(* IEC 61131-3 sources: F100R_S278_Temperville/MyController.device.xml.v3^/Plc Logic.plclogic.xml.v3^/Application.application.xml.v3^/07_Energia, 9 files *)

(* ---- C_ComposicaoFatura.prg.st ---- *)
PROGRAM C_ComposicaoFatura
VAR
	TonHabilita: TON;
	xTonHabilitaIn: BOOL;
	xTonHabilitaQ: BOOL;
	xTonHabilitaPt: TIME;
	PulsoLeitura: PulsoPositivo;
	PulsoLeituraIn: BOOL;
	PulsoLeituraQ: BOOL;
	xIntervaloPonta: BOOL;
	xIntervaloFPonta: BOOL;
	xIntervaloFPonta01: BOOL;
	xIntervaloFPonta02: BOOL;
	xFimMes: BOOL;
	xFechaConta: BOOL;
	rDemandaInstantaneaReal_kW: REAL;
END_VAR

(*LÓGICA DE COMPOSIÇÃO DA FATURA DE ENERGIA E ZERAMENTO DO MEDIDOR*)

// Dia da Leitura -> Fecha Fatura

IF uDiadaLeitura=uDiaRealTime THEN
	PulsoLeituraIn:=TRUE;
ELSE
	PulsoLeituraIn:=FALSE;
END_IF

PulsoLeitura(Entrada:=PulsoLeituraIn , SaidaPulsoPo=>PulsoLeituraQ );

IF PulsoLeituraQ THEN
	xFimMes:=TRUE;
END_IF

IF xFimMes THEN
	xFechaFatura:=1;
	xFimMes:=FALSE;
END_IF

(*-------------------------------------------------------------------------*)
xTonHabilitaIn:=TRUE;
TonHabilita(IN:=xTonHabilitaIn , PT:=T#300MS(*xTonHabilitaPt*) , Q=> xTonHabilitaQ, ET=> );

(*========= INTERVALOS DE PONTA E FORA PONTA =========*)

IF uHoraRealTime>=uHoraPonta  AND uHoraRealTime<=uHoraFPonta THEN
	xIntervaloPonta:=TRUE;
	xIntervaloFPonta:=FALSE;
ELSE
	xIntervaloFPonta:=TRUE;
	xIntervaloPonta:=FALSE;
END_IF

CASE PassoIntervalo OF
	//Seleção do Intervalo
		0: 	IF xIntervaloFPonta AND xTonHabilitaQ THEN
				PassoIntervalo:=5;
			END_IF
			IF xIntervaloPonta AND xTonHabilitaQ THEN
				PassoIntervalo:=50;
			END_IF
	// Consumos Fora Ponta
		5:	rConsumoInicialFPonta_kW:=rConsumoEnergiaReal_kWh;(*Ativo*)
			rConsumoInicialFPonta_kVAR:=rConsumoEnergiaReativa_kVARh;(*Reativo*)
			PassoIntervalo:=10;

		10:	rConsumoInstantaneoFPonta_kW:=rConsumoEnergiaReal_kWh-rConsumoInicialFPonta_kW;(*Ativo*)
			rConsumoInstantAcumFPonta_kW:=rConsumoAcumuladoFPonta_kW+rConsumoInstantaneoFPonta_kW;(*Ativo*)
			rConsumoInstantaneoFPonta_kVAR:=rConsumoEnergiaReativa_kVARh-rConsumoInicialFPonta_kVAR;(*Reativo*)
			rConsumoInstantAcumFPonta_kVAR:=rConsumoAcumuladoFPonta_kVAR+rConsumoInstantaneoFPonta_kVAR;(*Reativo*)

			rDemandaInstantaneaReal_kW:=rDemandaTotalReal_kW;
			IF rDemandaInstantaneaReal_kW>rDemandaMaximaPeriodo_kW THEN
				rDemandaMaximaPeriodo_kW:=rDemandaInstantaneaReal_kW;
			END_IF

			IF rDemandaTotalReal_kW>rDemandaMaximaIntervalo THEN
				rDemandaMaximaIntervalo:=rDemandaTotalReal_kW;
			END_IF

			IF NOT xIntervaloFPonta AND xTonHabilitaQ THEN
				PassoIntervalo:=15;
			END_IF
			IF (xFechaFatura=1) AND xTonHabilitaQ THEN
				PassoIntervalo:=16;
			END_IF

		15:	rConsumoAcumuladoFPonta_kW:=rConsumoInstantAcumFPonta_kW;(*Ativo*)
			rConsumoAcumuladoFPonta_kVAR:=rConsumoInstantAcumFPonta_kVAR;(*Reativo*)
			rConsumoFPonta_kW:=rConsumoInstantaneoFPonta_kW;(*Ativo*)
			rConsumoFPonta_kVAR:=rConsumoInstantaneoFPonta_kVAR;(*Reativo*)
			rDemandaMaxUltimoPeriodo:=rDemandaMaximaPeriodo_kW;
			PassoIntervalo:=16;

		16:	PassoIntervalo:=20;

		18: rConsumoAcumuladoFPonta_kW:=rConsumoInstantAcumFPonta_kW;(*Ativo*)
			rConsumoAcumuladoFPonta_kVAR:=rConsumoInstantAcumFPonta_kVAR;(*Reativo*)
			rConsumoFPonta_kW:=rConsumoInstantaneoFPonta_kW;(*Ativo*)
			rConsumoFPonta_kVAR:=rConsumoInstantaneoFPonta_kVAR;(*Reativo*)
			//rDemandaMaxUltimoIntervalo:=rDemandaMaximaReal_kW;
			rDemandaMaxUltimoIntervalo:=rDemandaMaximaIntervalo;
			PassoIntervalo:=20;

		20:	rConsumoInstantaneoFPonta_kW:=0;(*Ativo*)
			rConsumoInstantaneoFPonta_kVAR:=0;(*Reativo*)
			rDemandaMaximaPeriodo_kW:=0;
			IF (xFechaFatura=1) THEN
				xFechaConta:=TRUE;
			END_IF
			PassoIntervalo:=0;
	// Consumos Ponta
		50:	rConsumoInicialPonta_kW:=rConsumoEnergiaReal_kWh;(*Ativo*)
			rConsumoInicialPonta_kVAR:=rConsumoEnergiaReativa_kVARh;(*Reativo*)
			PassoIntervalo:=55;

		55:	rConsumoInstantaneoPonta_kW:=rConsumoEnergiaReal_kWh-rConsumoInicialPonta_kW;(*Ativo*)
			rConsumoInstantAcumPonta_kW:=rConsumoAcumuladoPonta_kW+rConsumoInstantaneoPonta_kW;(*Ativo*)
			rConsumoInstantaneoPonta_kVAR:=rConsumoEnergiaReativa_kVARh-rConsumoInicialPonta_kVAR;(*Reativo*)
			rConsumoInstantAcumPonta_kVAR:=rConsumoAcumuladoPonta_kVAR+rConsumoInstantaneoPonta_kVAR;(*Reativo*)

			rDemandaInstantaneaReal_kW:=rDemandaTotalReal_kW;
			IF rDemandaInstantaneaReal_kW>rDemandaMaximaPeriodo_kW THEN
				rDemandaMaximaPeriodo_kW:=rDemandaInstantaneaReal_kW;
			END_IF

			IF rDemandaTotalReal_kW>rDemandaMaximaIntervalo THEN
				rDemandaMaximaIntervalo:=rDemandaTotalReal_kW;
			END_IF

			IF NOT xIntervaloPonta AND xTonHabilitaQ THEN
				PassoIntervalo:=60;
			END_IF
			IF (xFechaFatura=1) AND xTonHabilitaQ THEN
				PassoIntervalo:=61;
			END_IF

		60:	rConsumoPonta_kW:=rConsumoInstantaneoPonta_kW;(*Ativo*)
			rConsumoAcumuladoPonta_kW:=rConsumoInstantAcumPonta_kW;(*Ativo*)
	      	rConsumoPonta_kVAR:=rConsumoInstantaneoPonta_kVAR;(*Reativo*)
			rConsumoAcumuladoPonta_kVAR:=rConsumoInstantAcumPonta_kVAR;(*Reativo*)
			rDemandaMaxUltimoPeriodo:=rDemandaMaximaPeriodo_kW;
			PassoIntervalo:=61;

		61:	PassoIntervalo:=65;

		63:	rConsumoPonta_kW:=rConsumoInstantaneoPonta_kW;(*Ativo*)
			rConsumoAcumuladoPonta_kW:=rConsumoInstantAcumPonta_kW;(*Ativo*)
	      	rConsumoPonta_kVAR:=rConsumoInstantaneoPonta_kVAR;(*Reativo*)
			rConsumoAcumuladoPonta_kVAR:=rConsumoInstantAcumPonta_kVAR;(*Reativo*)
			//rDemandaMaxUltimoIntervalo:=rDemandaMaximaReal_kW;
			rDemandaMaxUltimoIntervalo:=rDemandaMaximaIntervalo;
			PassoIntervalo:=65;

		65:	rConsumoInstantaneoPonta_kW:=0;(*Ativo*)
			rConsumoInstantaneoPonta_kVAR:=0;(*Reativo*)
			rDemandaMaximaPeriodo_kW:=0;
			IF (xFechaFatura=1) THEN
				xFechaConta:=TRUE;
			END_IF
			PassoIntervalo:=0;
END_CASE

// Fechamento da Tarifa Mensal
IF xFechaConta AND xTonHabilitaQ THEN
	 rEnergiaAtivaPonta_kWh			:=rConsumoAcumuladoPonta_kW;
	 rEnergiaAtivaFPonta_kWh		:=rConsumoAcumuladoFPonta_kW;
	 rEnergiaReativaPonta_kVar		:=rConsumoAcumuladoPonta_kVAR;
	 rEnergiaReativaFPonta_kVar		:=rConsumoAcumuladoFPonta_kVAR;
	 rDemandaEnergia_kW				:=rDemandaMaxUltimoIntervalo;
	 xFechaConta:=FALSE;
END_IF

IF xFaturaFechada=1 THEN // Vem do Supervisório
	bZeraAcumulado		:=TRUE;
	xCmdResetGeralPm	:=TRUE;
	xFaturaFechada		:=0;
END_IF

(*--------------------------------------------------------------------------------------------------------
(*--------------- Consumo Intervalo Diario -------*)
(*========= INTERVALOS FORA PONTA 01 e 02 =========*)

IF uMinutoRealTime>=0 AND uMinutoRealTime<=uMinutoPonta THEN
	xIntervaloFPonta01:=TRUE;
	xIntervaloFPonta02:=FALSE;
ELSIF uMinutoRealTime>=uMinutoFPonta AND  uMinutoRealTime<59 THEN
	xIntervaloFPonta02:=TRUE;
	xIntervaloFPonta01:=FALSE;
ELSIF uMinutoRealTime>=uMinutoPonta AND uMinutoRealTime<=uMinutoFPonta THEN
	xIntervaloFPonta01:=FALSE;
	xIntervaloFPonta02:=FALSE;
END_IF

CASE PassoIntervaloDia OF

		0: 	IF xIntervaloFPonta01 AND xTonHabilitaQ THEN
				PassoIntervaloDia:=5;
			END_IF
			IF xIntervaloFPonta02 AND xTonHabilitaQ THEN
				PassoIntervaloDia:=50;
			END_IF

		5:	rConsumoInicialFPonta01:=rConsumoEnergiaReal_kWh;
			PassoIntervaloDia:=10;

		10:	rConsumoInstantaneoFPonta01:=rConsumoEnergiaReal_kWh-rConsumoInicialFPonta01;
			rConsumoInstantDiarioFPonta:=rConsumoInstantaneoFPonta01;
			IF NOT xIntervaloFPonta01 AND xTonHabilitaQ THEN
				PassoIntervaloDia:=15;
			END_IF

		15:	rConsumoFPonta01:=rConsumoInstantaneoFPonta01;
			PassoIntervaloDia:=20;

		20:	rConsumoInstantaneoFPonta01:=0;
			PassoIntervaloDia:=0;

		50:	rConsumoInicialFPonta02:=rConsumoEnergiaReal_kWh;
			PassoIntervaloDia:=55;

		55:	rConsumoInstantaneoFPonta02:=rConsumoEnergiaReal_kWh-rConsumoInicialFPonta02;
			rConsumoInstantDiarioFPonta:=rConsumoFPonta01+rConsumoInstantaneoFPonta02;
			IF NOT xIntervaloFPonta02 AND xTonHabilitaQ THEN
				PassoIntervaloDia:=60;
			END_IF

		60:	rConsumoFPonta02:=rConsumoInstantaneoFPonta02;
			PassoIntervaloDia:=65;

		65:	rConsumoInstantaneoFPonta02:=0;
			rConsumoInstantDiarioFPonta:=0;
			PassoIntervaloDia:=70;

		70:	rConsumoDiarioFPonta:=rConsumoFPonta01+rConsumoFPonta02;
			rConsumoInicialFPonta01:=0;
			rConsumoInstantaneoFPonta01:=0;
			rConsumoFPonta01:=0;
			rConsumoInicialFPonta02:=0;
			rConsumoInstantaneoFPonta02:=0;
			rConsumoFPonta02:=0;
			PassoIntervaloDia:=0;

END_CASE
---------------------------------------------------------------------------------------------------------------*)
// ENERGIA CONSUMO DIÁRIO

rConsumoDiario:= rConsumoEnergiaReal_kWh-rConsumoDiarioInicial_kW;

IF	(uHoraRealTime=23 AND uMinutoRealTime=59 AND uSegundoRealTime=0) THEN
	rConsumoDiarioRel:=rConsumoDiario;
	xGrvRelatorioEnerg:=TRUE;

END_IF

IF	(uHoraRealTime=0 AND uMinutoRealTime=0 AND uSegundoRealTime=0)  THEN
	rConsumoDiarioInicial_kW:=rConsumoEnergiaReal_kWh;

END_IF

(* ---- D_ZeramentoMedidor.prg.st ---- *)
PROGRAM D_ZeramentoMedidor
VAR
	///Passo da Execução Reset Medidor de Energia
	PassoResetPm: INT;
	uResetValoresPM: UINT;
	xTriggerResetPM: BOOL;
	TonReset: TON;
	xTonResetIn: BOOL;
	xTonResetQ: BOOL;
	xTonResePt: TIME := TIME#2s0ms;
END_VAR

//Zeramento do Valores do Medidor
CASE PassoResetPm OF

		0:	IF xCmdResetGeralPm THEN
				uResetValoresPM:=14255;
				PassoResetPm:=1;
			END_IF

		1: IF uResetValoresPM=14255 THEN
				PassoResetPm:=3;
			END_IF

		3:	xTonResetIn:=TRUE;
			IF	xTonResetQ THEN
					PassoResetPm:=5;
			END_IF

		5:	xTonResetIn:=FALSE;
			xTriggerResetPM:=TRUE;
			PassoResetPm:=7;

		7:	xTonResetIn:=TRUE;
			IF	xTonResetQ THEN
					PassoResetPm:=10;
			END_IF

		10: xTonResetIn:=FALSE;
			xTriggerResetPM:=FALSE;
			uResetValoresPM:=30078;
			PassoResetPm:=11;

		11: IF uResetValoresPM=30078 THEN
				PassoResetPm:=13;
			END_IF

		13:	xTonResetIn:=TRUE;
			IF	xTonResetQ THEN
					PassoResetPm:=15;
			END_IF

		15:	xTonResetIn:=FALSE;
			xTriggerResetPM:=TRUE;
			PassoResetPm:=17;

		17:	xTonResetIn:=TRUE;
			IF	xTonResetQ AND rConsumoEnergiaReal_kWh=0 THEN
					PassoResetPm:=20;
			END_IF

		20:	xTonResetIn:=FALSE;
			xTriggerResetPM:=FALSE;
			uResetValoresPM:=21212;
			PassoResetPm:=21;

		21: IF uResetValoresPM=21212 THEN
				PassoResetPm:=23;
			END_IF

		23:	xTonResetIn:=TRUE;
			IF	xTonResetQ THEN
					PassoResetPm:=25;
			END_IF

		25:	xTonResetIn:=FALSE;
			xTriggerResetPM:=TRUE;
			PassoResetPm:=27;

		27:	xTonResetIn:=TRUE;
			IF	xTonResetQ THEN
					PassoResetPm:=30;
			END_IF

		30:	xTonResetIn:=FALSE;
			xTriggerResetPM:=FALSE;
			uResetValoresPM:=10001;
			PassoResetPm:=31;

		31: IF uResetValoresPM=10001 THEN
				PassoResetPm:=33;
			END_IF

		33:	xTonResetIn:=TRUE;
			IF	xTonResetQ THEN
					PassoResetPm:=35;
			END_IF

		35:	xTonResetIn:=FALSE;
			xTriggerResetPM:=TRUE;
			PassoResetPm:=37;

		37:	xTonResetIn:=TRUE;
			IF	xTonResetQ THEN
					PassoResetPm:=40;
			END_IF

		40:	xTonResetIn:=FALSE;
			xTriggerResetPM:=FALSE;
			uResetValoresPM:=0;
			bZeraAcumulado:=TRUE;
			xCmdResetGeralPm:=FALSE;
			PassoResetPm:=0;

END_CASE
TonReset(IN:= xTonResetIn, PT:=T#2S(*xTonResePt*) , Q=> xTonResetQ, ET=> );

// Zeramento das Memorias Acumuladas
IF bZeraAcumulado THEN
	PassoIntervalo				:=0;

	rConsumoInicialFPonta_kW	:=0;
	rConsumoInstantaneoFPonta_kW:=0;
	rConsumoFPonta_kW			:=0;
	rConsumoInstantAcumFPonta_kW:=0;
	rConsumoAcumuladoFPonta_kW	:=0;

	rConsumoInicialPonta_kW		:=0;
	rConsumoInstantaneoPonta_kW	:=0;
	rConsumoPonta_kW			:=0;
	rConsumoInstantAcumPonta_kW	:=0;
	rConsumoAcumuladoPonta_kW	:=0;

	rConsumoInicialFPonta_kVAR	:=0;
	rConsumoInstantaneoFPonta_kVAR:=0;
	rConsumoFPonta_kVAR			:=0;
	rConsumoInstantAcumFPonta_kVAR:=0;
	rConsumoAcumuladoFPonta_kVAR:=0;

	rConsumoInicialPonta_kVAR	:=0;
	rConsumoInstantaneoPonta_kVAR:=0;
	rConsumoPonta_kVAR			:=0;
	rConsumoInstantAcumPonta_kVAR:=0;
	rConsumoAcumuladoPonta_kVAR	:=0;

//	rConsumoInicialFPonta01		:=0;
//	rConsumoInstantaneoFPonta01	:=0;
//	rConsumoFPonta01			:=0;

//	rConsumoInicialFPonta02		:=0;
//	rConsumoInstantaneoFPonta02	:=0;
//	rConsumoFPonta02			:=0;

	rConsumoDiarioFPonta		:=0;
	//xFaturaFechada				:=0;
	bZeraAcumulado				:=FALSE;
END_IF

(* ---- E_Nobreak.prg.st ---- *)
PROGRAM E_Nobreak
VAR
	TonNobreak: TON;
	TonNobreakIn: BOOL;
	TonNobreakQ: BOOL;
	TpSonAlmNbk: TP;
END_VAR

xStatusNobreak:=xSaidaNobreakOk;

TonNobreakIn:= NOT xSaidaNobreakOk;
TonNobreak(IN:=TonNobreakIn , PT:=T#500MS , Q=>TonNobreakQ , ET=> );
IF TonNobreakQ THEN
	xAlmNobreak:=TRUE;
END_IF

TpSonAlmNbk(IN:=xAlmNobreak , PT:=T#500MS , Q=> , ET=> );

IF TpSonAlmNbk.Q THEN
	xAlmNobreakSom:=TRUE;
END_IF

IF	bResetAlmGeral THEN
	xAlmNobreak:=FALSE;
	xAlmNobreakSom:=FALSE;
END_IF

xNobreakDesabilitado:= NOT xNobreakHabilitado;

(* ---- Energia.prg.st ---- *)
PROGRAM Energia
VAR
	Double01: WORD_AS_DWORD;
	Double02: WORD_AS_DWORD;
	Double03: WORD_AS_DWORD;
	////////////////////////////////////////////////////////////////
	dConsumoEnergiaReal_kWh: DWORD;
	dConsumoEnergiaAparente_kVAh: DWORD;
	dConsumoEnergiaReativa_kVARh: DWORD;
	u0ConsumoEnergiaReal_kWh: WORD;
	u1ConsumoEnergiaReal_kWh: WORD;
	u0ConsumoEnergiaAparente_kVAh: WORD;
	u1ConsumoEnergiaAparente_kVAh: WORD;
	u0ConsumoEnergiaReativa_kVARh: WORD;
	u1ConsumoEnergiaReativa_kVARh: WORD;
	uPotenciaTotalReal_kW: UINT;
	uPotenciaTotalAparente_kVA: UINT;
	uPotenciaTotalReativa_kVAR: UINT;
	uFatorDePotenciaTotal: UINT;
	uTensaoFFMedia_V: UINT;
	uTensaoFNMedia_V: UINT;
	uCorrenteMedia_V: UINT;
	uFrequencia_Hz: UINT;
	uDemandaTotalReal_kW: UINT;
	uDemandaTotalAparente_kVA: UINT;
	uDemandaTotalReativa_kVAR: UINT;
	uDemandaMaximaReal_kW: UINT;
	uDemandaMaximaAparente_kVA: UINT;
	uDemandaMaximaReativa_kVAR: UINT;
	uCorrenteInstantFaseA_Amp: UINT;
	uCorrenteInstantFaseB_Amp: UINT;
	uCorrenteInstantFaseC_Amp: UINT;
	uCorrenteInstantNeutro_Amp: UINT;
	uCorrenteDemandaFaseA_Amp: UINT;
	uCorrenteDemandaFaseB_Amp: UINT;
	uCorrenteDemandaFaseC_Amp: UINT;
	uCorrenteMaximaDemandaFaseA_Amp: UINT;
	uCorrenteMaximaDemandaFaseB_Amp: UINT;
	uCorrenteMaximaDemandaFaseC_Amp: UINT;
	uTensaoFaseAB_V: UINT;
	uTensaoFaseBC_V: UINT;
	uTensaoFaseAC_V: UINT;
	uTensaoFaseAN_V: UINT;
	uTensaoFaseBN_V: UINT;
	uTensaoFaseCN_V: UINT;
	uPotenciaRealFaseA_kW: UINT;
	uPotenciaRealFaseB_kW: UINT;
	uPotenciaRealFaseC_kW: UINT;
	uPotenciaAparenteFaseA_kVA: UINT;
	uPotenciaAparenteFaseB_kVA: UINT;
	uPotenciaAparenteFaseC_kVA: UINT;
	uPotenciaReativaFaseA_kVAR: UINT;
	uPotenciaReativaFaseB_kVAR: UINT;
	uPotenciaReativaFaseC_kVAR: UINT;
	uCorrenteTHDFaseA: UINT;
	uCorrenteTHDFaseB: UINT;
	uCorrenteTHDFaseC: UINT;
	uCorrenteTHDNeutro: UINT;
	uTensaoTHDFaseAN: UINT;
	uTensaoTHDFaseBN: UINT;
	uTensaoTHDFaseCN: UINT;
	uTensaoTHDFaseAB: UINT;
	uTensaoTHDFaseBC: UINT;
	uTensaoTHDFaseAC: UINT;
	/// Valores minimos
	uPotenciaTotalRealMinima_kW: UINT;
	uPotenciaTotalAparenteMinima_kVA: UINT;
	uPotenciaTotalReativaMinima_kVAR: UINT;
	uFatorDePotenciaTotalMinima: UINT;
	uFrequenciaMinima_Hz: UINT;
	uCorrenteMinimaFaseA_Amp: UINT;
	uCorrenteMinimaFaseB_Amp: UINT;
	uCorrenteMinimaFaseC_Amp: UINT;
	uCorrenteMinimaNeutro_Amp: UINT;
	uTensaoMinimaFaseAN_V: UINT;
	uTensaoMinimaFaseBN_V: UINT;
	uTensaoMinimaFaseCN_V: UINT;
	uTensaoMinimaFaseAB_V: UINT;
	uTensaoMinimaFaseBC_V: UINT;
	uTensaoMinimaFaseAC_V: UINT;
	uCorrenteTHDMinimoFaseA: UINT;
	uCorrenteTHDMinimoFaseB: UINT;
	uCorrenteTHDMinimoFaseC: UINT;
	uCorrenteTHDMinimoNeutro: UINT;
	uTensaoTHDMinimoFaseAN: UINT;
	uTensaoTHDMinimoFaseBN: UINT;
	uTensaoTHDMinimoFaseCN: UINT;
	uTensaoTHDMinimoFaseAB: UINT;
	uTensaoTHDMinimoFaseBC: UINT;
	uTensaoTHDMinimoFaseAC: UINT;
	/// Valores Maximos
	uPotenciaTotalRealMaximo_kW: UINT;
	uPotenciaTotalAparenteMaximo_kVA: UINT;
	uPotenciaTotalReativaMaximo_kVAR: UINT;
	uFatorDePotenciaTotalMaximo: UINT;
	uFrequenciaMaxima_Hz: UINT;
	uCorrenteMaximoFaseA_Amp: UINT;
	uCorrenteMaximoFaseB_Amp: UINT;
	uCorrenteMaximoFaseC_Amp: UINT;
	uCorrenteMaximoNeutro_Amp: UINT;
	uTensaoMaximoFaseAN_V: UINT;
	uTensaoMaximoFaseBN_V: UINT;
	uTensaoMaximoFaseCN_V: UINT;
	uTensaoMaximoFaseAB_V: UINT;
	uTensaoMaximoFaseBC_V: UINT;
	uTensaoMaximoFaseAC_V: UINT;
	uCorrenteTHDMaximoFaseA: UINT;
	uCorrenteTHDMaximoFaseB: UINT;
	uCorrenteTHDMaximoFaseC: UINT;
	uCorrenteTHDMaximoNeutro: UINT;
	uTensaoTHDMaximoFaseAN: UINT;
	uTensaoTHDMaximoFaseBN: UINT;
	uTensaoTHDMaximoFaseCN: UINT;
	uTensaoTHDMaximoFaseAB: UINT;
	uTensaoTHDMaximoFaseBC: UINT;
	uTensaoTHDMaximoFaseAC: UINT;
END_VAR

Double01(i_wLow:= u1ConsumoEnergiaReal_kWh, i_wHigh:= u0ConsumoEnergiaReal_kWh, q_dwOput=> dConsumoEnergiaReal_kWh);
Double02(i_wLow:= u1ConsumoEnergiaAparente_kVAh, i_wHigh:= u0ConsumoEnergiaAparente_kVAh, q_dwOput=> dConsumoEnergiaAparente_kVAh);
Double03(i_wLow:= u1ConsumoEnergiaReativa_kVARh, i_wHigh:= u0ConsumoEnergiaReativa_kVARh, q_dwOput=> dConsumoEnergiaReativa_kVARh);

rConsumoEnergiaReal_kWh			:=fEnergiaAtivaAcumulada/1000;//(DINT_TO_REAL(DWORD_TO_DINT(dConsumoEnergiaReal_kWh)))/10;
rConsumoEnergiaAparente_kVAh	:=fEnergiaAparenteAcumulada/1000;//(DINT_TO_REAL(DWORD_TO_DINT(dConsumoEnergiaAparente_kVAh)))/10;
rConsumoEnergiaReativa_kVARh	:=fEnergiaReativaAcumulada/1000;//(DINT_TO_REAL(DWORD_TO_DINT(dConsumoEnergiaReativa_kVARh)))/10;
rPotenciaTotalReal_kW			:=fPotenciaAtivaTotal;//(INT_TO_REAL(UINT_TO_INT(uPotenciaTotalReal_kW)));
rPotenciaTotalAparente_kVA		:=(INT_TO_REAL(UINT_TO_INT(uPotenciaTotalAparente_kVA)));
rPotenciaTotalReativa_kVAR 		:=(INT_TO_REAL(UINT_TO_INT(uPotenciaTotalReativa_kVAR)))/10;
rFatorDePotenciaTotal 			:=fFatorPotenciaTotal;//(INT_TO_REAL(UINT_TO_INT(uFatorDePotenciaTotal)))/10000;
rTensaoFFMedia_V				:=fTensaoAvgLL;//(INT_TO_REAL(UINT_TO_INT(uTensaoFFMedia_V)))/10;
rTensaoFNMedia_V				:=fTensaoAvgLN;//(INT_TO_REAL(UINT_TO_INT(uTensaoFNMedia_V)))/10;
rCorrenteMedia_V				:=fCorrenteAvg;//(INT_TO_REAL(UINT_TO_INT(uCorrenteMedia_V)));
rFrequencia_Hz					:=fFrequencia;//(INT_TO_REAL(UINT_TO_INT(uFrequencia_Hz)))/100;
rDemandaTotalReal_kW			:=fUltimaDemanda;//(INT_TO_REAL(UINT_TO_INT(uDemandaTotalReal_kW)));
rDemandaTotalAparente_kVA		:=(INT_TO_REAL(UINT_TO_INT(uDemandaTotalAparente_kVA)));
rDemandaTotalReativa_kVAR		:=(INT_TO_REAL(UINT_TO_INT(uDemandaTotalReativa_kVAR)))/10;
rDemandaMaximaReal_kW			:=fPicoDemanda;//(INT_TO_REAL(UINT_TO_INT(uDemandaMaximaReal_kW)));
rDemandaMaximaAparente_kVA		:=(INT_TO_REAL(UINT_TO_INT(uDemandaMaximaAparente_kVA)))/10;
rDemandaMaximaReativa_kVAR		:=(INT_TO_REAL(UINT_TO_INT(uDemandaMaximaReativa_kVAR)))/10;
rCorrenteInstantFaseA_Amp		:=fCorrenteFaseA;//(INT_TO_REAL(UINT_TO_INT(uCorrenteInstantFaseA_Amp)))/1;
rCorrenteInstantFaseB_Amp 		:=fCorrenteFaseB;//(INT_TO_REAL(UINT_TO_INT(uCorrenteInstantFaseB_Amp)))/1;
rCorrenteInstantFaseC_Amp 		:=fCorrenteFaseC;//(INT_TO_REAL(UINT_TO_INT(uCorrenteInstantFaseC_Amp)))/1;
rCorrenteInstantNeutro_Amp 		:=fCorrenteNeutro;//(INT_TO_REAL(UINT_TO_INT(uCorrenteInstantNeutro_Amp)))/1;
rCorrenteDemandaFaseA_Amp		:=(INT_TO_REAL(UINT_TO_INT(uCorrenteDemandaFaseA_Amp)))/10;
rCorrenteDemandaFaseB_Amp		:=(INT_TO_REAL(UINT_TO_INT(uCorrenteDemandaFaseB_Amp)))/10;
rCorrenteDemandaFaseC_Amp		:=(INT_TO_REAL(UINT_TO_INT(uCorrenteDemandaFaseC_Amp)))/10;
rCorrenteMaximaDemandaFaseA_Amp	:=(INT_TO_REAL(UINT_TO_INT(uCorrenteMaximaDemandaFaseA_Amp)))/10;
rCorrenteMaximaDemandaFaseB_Amp	:=(INT_TO_REAL(UINT_TO_INT(uCorrenteMaximaDemandaFaseB_Amp)))/10;
rCorrenteMaximaDemandaFaseC_Amp	:=(INT_TO_REAL(UINT_TO_INT(uCorrenteMaximaDemandaFaseC_Amp)))/10;
rTensaoFaseAB_V					:=fTensaoAB;//(INT_TO_REAL(UINT_TO_INT(uTensaoFaseAB_V)))/10;
rTensaoFaseBC_V					:=fTensaoBC;//(INT_TO_REAL(UINT_TO_INT(uTensaoFaseBC_V)))/10;
rTensaoFaseAC_V					:=fTensaoCA;//(INT_TO_REAL(UINT_TO_INT(uTensaoFaseAC_V)))/10;
rTensaoFaseAN_V					:=fTensaoAN;//(INT_TO_REAL(UINT_TO_INT(uTensaoFaseAN_V)))/10;
rTensaoFaseBN_V					:=fTensaoBN;//(INT_TO_REAL(UINT_TO_INT(uTensaoFaseBN_V)))/10;
rTensaoFaseCN_V					:=fTensaoCN;//(INT_TO_REAL(UINT_TO_INT(uTensaoFaseCN_V)))/10;
rPotenciaRealFaseA_kW			:=(INT_TO_REAL(UINT_TO_INT(uPotenciaRealFaseA_kW)))/10;
rPotenciaRealFaseB_kW			:=(INT_TO_REAL(UINT_TO_INT(uPotenciaRealFaseB_kW)))/10;
rPotenciaRealFaseC_kW			:=(INT_TO_REAL(UINT_TO_INT(uPotenciaRealFaseC_kW)))/10;
rPotenciaAparenteFaseA_kVA		:=(INT_TO_REAL(UINT_TO_INT(uPotenciaAparenteFaseA_kVA)))/10;
rPotenciaAparenteFaseB_kVA		:=(INT_TO_REAL(UINT_TO_INT(uPotenciaAparenteFaseB_kVA)))/10;
rPotenciaAparenteFaseC_kVA		:=(INT_TO_REAL(UINT_TO_INT(uPotenciaAparenteFaseC_kVA)))/10;
rPotenciaReativaFaseA_kVAR		:=(INT_TO_REAL(UINT_TO_INT(uPotenciaReativaFaseA_kVAR)))/10;
rPotenciaReativaFaseB_kVAR		:=(INT_TO_REAL(UINT_TO_INT(uPotenciaReativaFaseB_kVAR)))/10;
rPotenciaReativaFaseC_kVAR		:=(INT_TO_REAL(UINT_TO_INT(uPotenciaReativaFaseC_kVAR)))/10;
rCorrenteTHDFaseA				:=(INT_TO_REAL(UINT_TO_INT(uCorrenteTHDFaseA)))/10;
rCorrenteTHDFaseB				:=(INT_TO_REAL(UINT_TO_INT(uCorrenteTHDFaseB)))/10;
rCorrenteTHDFaseC				:=(INT_TO_REAL(UINT_TO_INT(uCorrenteTHDFaseC)))/10;
rCorrenteTHDNeutro				:=(INT_TO_REAL(UINT_TO_INT(uCorrenteTHDNeutro)))/10;
rTensaoTHDFaseAN				:=(INT_TO_REAL(UINT_TO_INT(uTensaoTHDFaseAN)))/10;
rTensaoTHDFaseBN				:=(INT_TO_REAL(UINT_TO_INT(uTensaoTHDFaseBN)))/10;
rTensaoTHDFaseCN				:=(INT_TO_REAL(UINT_TO_INT(uTensaoTHDFaseCN)))/10;
rTensaoTHDFaseAB				:=(INT_TO_REAL(UINT_TO_INT(uTensaoTHDFaseAB)))/10;
rTensaoTHDFaseBC				:=(INT_TO_REAL(UINT_TO_INT(uTensaoTHDFaseBC)))/10;
rTensaoTHDFaseAC				:=(INT_TO_REAL(UINT_TO_INT(uTensaoTHDFaseAC)))/10;

// Valores minimos

rPotenciaTotalRealMinima_kW 	:=(INT_TO_REAL(UINT_TO_INT(uPotenciaTotalRealMinima_kW)))/10;
rPotenciaTotalAparenteMinima_kVA:=(INT_TO_REAL(UINT_TO_INT(uPotenciaTotalAparenteMinima_kVA)))/10;
rPotenciaTotalReativaMinima_kVAR:=(INT_TO_REAL(UINT_TO_INT(uPotenciaTotalReativaMinima_kVAR)))/10;
rFatorDePotenciaTotalMinima 	:=(INT_TO_REAL(UINT_TO_INT(uFatorDePotenciaTotalMinima)))/10;
rFrequenciaMinima_Hz			:=(INT_TO_REAL(UINT_TO_INT(uFrequenciaMinima_Hz)))/10;
rCorrenteMinimaFaseA_Amp 		:=(INT_TO_REAL(UINT_TO_INT(uCorrenteMinimaFaseA_Amp)))/10;
rCorrenteMinimaFaseB_Amp 		:=(INT_TO_REAL(UINT_TO_INT(uCorrenteMinimaFaseB_Amp)))/10;
rCorrenteMinimaFaseC_Amp 		:=(INT_TO_REAL(UINT_TO_INT(uCorrenteMinimaFaseC_Amp)))/10;
rCorrenteMinimaNeutro_Amp 		:=(INT_TO_REAL(UINT_TO_INT(uCorrenteMinimaNeutro_Amp)))/10;
rTensaoMinimaFaseAN_V			:=(INT_TO_REAL(UINT_TO_INT(uTensaoMinimaFaseAN_V)))/10;
rTensaoMinimaFaseBN_V			:=(INT_TO_REAL(UINT_TO_INT(uTensaoMinimaFaseBN_V)))/10;
rTensaoMinimaFaseCN_V			:=(INT_TO_REAL(UINT_TO_INT(uTensaoMinimaFaseCN_V)))/10;
rTensaoMinimaFaseAB_V			:=(INT_TO_REAL(UINT_TO_INT(uTensaoMinimaFaseAB_V)))/10;
rTensaoMinimaFaseBC_V			:=(INT_TO_REAL(UINT_TO_INT(uTensaoMinimaFaseBC_V)))/10;
rTensaoMinimaFaseAC_V			:=(INT_TO_REAL(UINT_TO_INT(uTensaoMinimaFaseAC_V)))/10;
rCorrenteTHDMinimoFaseA			:=(INT_TO_REAL(UINT_TO_INT(uCorrenteTHDMinimoFaseA)))/10;
rCorrenteTHDMinimoFaseB			:=(INT_TO_REAL(UINT_TO_INT(uCorrenteTHDMinimoFaseB)))/10;
rCorrenteTHDMinimoFaseC			:=(INT_TO_REAL(UINT_TO_INT(uCorrenteTHDMinimoFaseC)))/10;
rCorrenteTHDMinimoNeutro		:=(INT_TO_REAL(UINT_TO_INT(uCorrenteTHDMinimoNeutro)))/10;
rTensaoTHDMinimoFaseAN			:=(INT_TO_REAL(UINT_TO_INT(uTensaoTHDMinimoFaseAN)))/10;
rTensaoTHDMinimoFaseBN			:=(INT_TO_REAL(UINT_TO_INT(uTensaoTHDMinimoFaseBN)))/10;
rTensaoTHDMinimoFaseCN			:=(INT_TO_REAL(UINT_TO_INT(uTensaoTHDMinimoFaseCN)))/10;
rTensaoTHDMinimoFaseAB			:=(INT_TO_REAL(UINT_TO_INT(uTensaoTHDMinimoFaseAB)))/10;
rTensaoTHDMinimoFaseBC			:=(INT_TO_REAL(UINT_TO_INT(uTensaoTHDMinimoFaseBC)))/10;
rTensaoTHDMinimoFaseAC			:=(INT_TO_REAL(UINT_TO_INT(uTensaoTHDMinimoFaseAC)))/10;

// Valores Maximos

rPotenciaTotalRealMaximo_kW 	:=(INT_TO_REAL(UINT_TO_INT(uPotenciaTotalRealMaximo_kW)))/10;
rPotenciaTotalAparenteMaximo_kVA:=(INT_TO_REAL(UINT_TO_INT(uPotenciaTotalAparenteMaximo_kVA)))/10;
rPotenciaTotalReativaMaximo_kVAR:=(INT_TO_REAL(UINT_TO_INT(uPotenciaTotalReativaMaximo_kVAR)))/10;
rFatorDePotenciaTotalMaximo 	:=(INT_TO_REAL(UINT_TO_INT(uFatorDePotenciaTotalMaximo)))/10;
rFrequenciaMaxima_Hz			:=(INT_TO_REAL(UINT_TO_INT(uFrequenciaMaxima_Hz)))/10;
rCorrenteMaximoFaseA_Amp 		:=fCorrenteMaximaFaseA;//(INT_TO_REAL(UINT_TO_INT(uCorrenteMaximoFaseA_Amp)))/10;
rCorrenteMaximoFaseB_Amp 		:=fCorrenteMaximaFaseB;//(INT_TO_REAL(UINT_TO_INT(uCorrenteMaximoFaseB_Amp)))/10;
rCorrenteMaximoFaseC_Amp 		:=fCorrenteMaximaFaseC;//(INT_TO_REAL(UINT_TO_INT(uCorrenteMaximoFaseC_Amp)))/10;
rCorrenteMaximoNeutro_Amp 		:=fCorrenteMaximaNeutro;//(INT_TO_REAL(UINT_TO_INT(uCorrenteMaximoNeutro_Amp)))/10;
rTensaoMaximoFaseAN_V			:=fTensaoMaximaAN;//(INT_TO_REAL(UINT_TO_INT(uTensaoMaximoFaseAN_V)))/10;
rTensaoMaximoFaseBN_V			:=fTensaoMaximaAN;//(INT_TO_REAL(UINT_TO_INT(uTensaoMaximoFaseBN_V)))/10;
rTensaoMaximoFaseCN_V			:=fTensaoMaximaAN;//(INT_TO_REAL(UINT_TO_INT(uTensaoMaximoFaseCN_V)))/10;
rTensaoMaximoFaseAB_V			:=fTensaoMaximaAB;//(INT_TO_REAL(UINT_TO_INT(uTensaoMaximoFaseAB_V)))/10;
rTensaoMaximoFaseBC_V			:=fTensaoMaximaBC;//(INT_TO_REAL(UINT_TO_INT(uTensaoMaximoFaseBC_V)))/10;
rTensaoMaximoFaseAC_V			:=fTensaoMaximaCA;//(INT_TO_REAL(UINT_TO_INT(uTensaoMaximoFaseAC_V)))/10;
rCorrenteTHDMaximoFaseA			:=(INT_TO_REAL(UINT_TO_INT(uCorrenteTHDMaximoFaseA)))/10;
rCorrenteTHDMaximoFaseB			:=(INT_TO_REAL(UINT_TO_INT(uCorrenteTHDMaximoFaseB)))/10;
rCorrenteTHDMaximoFaseC			:=(INT_TO_REAL(UINT_TO_INT(uCorrenteTHDMaximoFaseC)))/10;
rCorrenteTHDMaximoNeutro		:=(INT_TO_REAL(UINT_TO_INT(uCorrenteTHDMaximoNeutro)))/10;
rTensaoTHDMaximoFaseAN			:=(INT_TO_REAL(UINT_TO_INT(uTensaoTHDMaximoFaseAN)))/10;
rTensaoTHDMaximoFaseBN			:=(INT_TO_REAL(UINT_TO_INT(uTensaoTHDMaximoFaseBN)))/10;
rTensaoTHDMaximoFaseCN			:=(INT_TO_REAL(UINT_TO_INT(uTensaoTHDMaximoFaseCN)))/10;
rTensaoTHDMaximoFaseAB			:=(INT_TO_REAL(UINT_TO_INT(uTensaoTHDMaximoFaseAB)))/10;
rTensaoTHDMaximoFaseBC			:=(INT_TO_REAL(UINT_TO_INT(uTensaoTHDMaximoFaseBC)))/10;
rTensaoTHDMaximoFaseAC			:=(INT_TO_REAL(UINT_TO_INT(uTensaoTHDMaximoFaseAC)))/10;

////////////////////////////////////////////////////////////////////////

(* ---- F_FaltaFase.prg.st ---- *)
PROGRAM F_FaltaFase
VAR
	xFaltaFaseA: BOOL;
	xFaltaFaseB: BOOL;
	xFaltaFaseC: BOOL;
	TpSemEnergia: TP;
	TonSemEnergia: TON;
	TonSemEnergiaIn: BOOL;
	TonSemEnergiaQ: BOOL;
	Tp02SemEnergia: TP;
END_VAR

IF rTensaoFaseAN_V<=190 THEN
	xFaltaFaseA:=TRUE;
ELSE
	xFaltaFaseA:=FALSE;
END_IF
IF rTensaoFaseBN_V<=190 THEN
	xFaltaFaseB:=TRUE;
ELSE
	xFaltaFaseB:=FALSE;
END_IF
IF rTensaoFaseCN_V<=190 THEN
	xFaltaFaseC:=TRUE;
ELSE
	xFaltaFaseC:=FALSE;
END_IF

IF xFaltaFaseA or xFaltaFaseB or xFaltaFaseC THEN
	TonSemEnergiaIn:=TRUE;
ELSE
	TonSemEnergiaIn:=FALSE;
END_IF

TonSemEnergia(IN:=TonSemEnergiaIn , PT:=T#1S , Q=>TonSemEnergiaQ , ET=> );

IF TonSemEnergiaQ THEN
	xSemEnergia:=TRUE;
	xEnergiaOk:=FALSE;
ELSE
	xSemEnergia:=FALSE;
	xEnergiaOk:=TRUE;
END_IF

TpSemEnergia(IN:=xSemEnergia , PT:=T#500MS , Q=> , ET=> );

IF TpSemEnergia.Q THEN
	xAlmSomSemEnergia:=TRUE;
END_IF

IF bResetAlmGeral THEN
	xAlmSomSemEnergia:=FALSE;
END_IF

TpSemEnergia(IN:=xSemEnergia , PT:=T#30S , Q=>xSomSemEnergia , ET=> );

(* ---- G_Disjuntores.prg.st ---- *)
PROGRAM G_Disjuntores
VAR
	TonDisjGeral: TON;
	TonDisjGeralIn: BOOL;
	TonDisjGeralQ: BOOL;
	TpSonAlmDisjGeral: TP;
	TonDisjResist: TON;
	TonDisjResistIn: BOOL;
	TonDisjResistQ: BOOL;
	TpSonAlmTonDisjResist: TP;
END_VAR

// MOITORAMENTO DO DISJUNTOR GERAL DO PAINEL
xDisjGeralOff:= NOT xDisjGeralOn;

TonDisjGeralIn:= xDisjGeralOff;
TonDisjGeral(IN:=TonDisjGeralIn , PT:=T#1000MS , Q=>TonDisjGeralQ , ET=> );
IF TonDisjGeralQ THEN
	xAlmDisjGeral:=TRUE;
END_IF

TpSonAlmDisjGeral(IN:=xAlmDisjGeral , PT:=T#500MS , Q=> , ET=> );

IF TpSonAlmDisjGeral.Q THEN
	xAlmDisjGeralSom:=TRUE;
END_IF

IF	bResetAlmGeral THEN
	xAlmDisjGeral:=FALSE;
	xAlmDisjGeralSom:=FALSE;
END_IF

// MONITORAMENTO DO DISJUNTOR GERAL DAS RESISTÊNCIAS
TonDisjResistIn:= xDisjResistOff AND xResistenciasLigadas;
TonDisjGeral(IN:=TonDisjResistIn , PT:=T#1000MS , Q=>TonDisjResistQ , ET=> );
IF TonDisjResistQ THEN
	xAlmDisjResist:=TRUE;
END_IF

TpSonAlmTonDisjResist(IN:=xAlmDisjResist , PT:=T#500MS , Q=> , ET=> );

IF TpSonAlmTonDisjResist.Q THEN
	xAlmDisjResistSom:=TRUE;
END_IF

IF	bResetAlmGeral THEN
	xAlmDisjResist:=FALSE;
	xAlmDisjResistSom:=FALSE;
END_IF

(* ---- H_CircuitoCC.prg.st ---- *)
PROGRAM H_CircuitoCC
VAR
END_VAR

// Habilita/Desabilita Circuito CC
xHabDesabCircuitoCC:= xChHabDesabCircuitoCC;

// Posição da Chave Liga Motores CC
xCircuitoEmergenciaCC:= NOT xChCircuitoEmergenciaCC;// AND xHabDesabCircuitoCC;

IF xMaquinaEmEspera AND xChCircuitoEmergenciaCC AND xHabDesabCircuitoCC THEN
	xAlertaPosChCircCC:= TRUE;
ELSE
	xAlertaPosChCircCC:= FALSE;
END_IF

(* ---- PM5300.prg.st ---- *)
PROGRAM PM5300
VAR
	/// 2999
	wCorrenteFaseA_W1: WORD;
	/// 3000
	wCorrenteFaseA_W0: WORD;
	/// 3001
	wCorrenteFaseB_W1: WORD;
	/// 3002
	wCorrenteFaseB_W0: WORD;
	/// 3003
	wCorrenteFaseC_W1: WORD;
	/// 3004
	wCorrenteFaseC_W0: WORD;
	/// 3005
	wCorrenteNeutro_W1: WORD;
	/// 3006
	wCorrenteNeutro_W0: WORD;
	/// 3007
	wCorrenteG_W1: WORD;
	/// 3008
	wCorrenteG_W0: WORD;
	/// 3009
	wCorrenteAvg_W1: WORD;
	/// 3010
	wCorrenteAvg_W0: WORD;
	/// 3019
	wTensaoAB_W1: WORD;
	/// 3020
	wTensaoAB_W0: WORD;
	/// 3021
	wTensaoBC_W1: WORD;
	/// 3022
	wTensaoBC_W0: WORD;
	/// 3023
	wTensaoCA_W1: WORD;
	/// 3024
	wTensaoCA_W0: WORD;
	/// 3025
	wTensaoAvgL_W1: WORD;
	/// 3026
	wTensaoAvgL_W0: WORD;
	/// 3027
	wTensaoAN_W1: WORD;
	/// 3028
	wTensaoAN_W0: WORD;
	/// 3029
	wTensaoBN_W1: WORD;
	/// 3030
	wTensaoBN_W0: WORD;
	/// 3031
	wTensaoCN_W1: WORD;
	/// 3032
	wTensaoCN_W0: WORD;
	/// 3035
	wTensaoAvgN_W1: WORD;
	/// 3036
	wTensaoAvgN_W0: WORD;
	///3059
	wPotenciaAtivaTotal_W1: WORD;
	///3060
	wPotenciaAtivaTotal_W0: WORD;
	///3083
	wFatorPotenciaTotal_W1: WORD;
	///3084
	wFatorPotenciaTotal_W0: WORD;
	///3109
	wFrequencia_W1: WORD;
	///3110
	wFrequencia_W0: WORD;
	///3762
	wUltimaDemanda_W1: WORD;
	///3763
	wUltimaDemanda_W0: WORD;
	///3764
	wAtualDemanda_W1: WORD;
	///3765
	wAtualDemanda_W0: WORD;
	///3766
	wPrevisaoDemanda_W1: WORD;
	///3767
	wPrevisaoDemanda_W0: WORD;
	///3768
	wPicoDemanda_W1: WORD;
	///3769
	wPicoDemanda_W0: WORD;
	///3203
	wEnergiaAtivaAcumulada_W1_High: WORD;
	///3204
	wEnergiaAtivaAcumulada_W0_High: WORD;
	///3205
	wEnergiaAtivaAcumulada_W1_Low: WORD;
	///3206
	wEnergiaAtivaAcumulada_W0_Low: WORD;
	///3219
	wEnergiaReativaAcumulada_W1_High: WORD;
	///3220
	wEnergiaReativaAcumulada_W0_High: WORD;
	///3221
	wEnergiaReativaAcumulada_W1_Low: WORD;
	///3222
	wEnergiaReativaAcumulada_W0_Low: WORD;
	///3235
	wEnergiaAparenteAcumulada_W1_High: WORD;
	///3236
	wEnergiaAparenteAcumulada_W0_High: WORD;
	///3237
	wEnergiaAparenteAcumulada_W1_Low: WORD;
	///3238
	wEnergiaAparenteAcumulada_W0_Low: WORD;
	lEnergiaAtivaAcumulada: LINT;
	lEnergiaReativaAcumulada: LINT;
	lEnergiaAparenteAcumulada: LINT;
	/// 27693
	wCorrenteMaximaFaseA_W1: WORD;
	wCorrenteMaximaFaseA_W0: WORD;
	wCorrenteMaximaFaseB_W1: WORD;
	wCorrenteMaximaFaseB_W0: WORD;
	wCorrenteMaximaFaseC_W1: WORD;
	wCorrenteMaximaFaseC_W0: WORD;
	wCorrenteMaximaNeutro_W1: WORD;
	wCorrenteMaximaNeutro_W0: WORD;
	wCorrenteMaximaG_W1: WORD;
	wCorrenteMaximaG_W0: WORD;
	wCorrenteMaximaAvg_W1: WORD;
	wCorrenteMaximaAvg_W0: WORD;
	wTensaoMaximaAB_W1: WORD;
	wTensaoMaximaAB_W0: WORD;
	wTensaoMaximaBC_W1: WORD;
	wTensaoMaximaBC_W0: WORD;
	wTensaoMaximaCA_W1: WORD;
	wTensaoMaximaCA_W0: WORD;
	wTensaoMaximaAvgL_W1: WORD;
	wTensaoMaximaAvgL_W0: WORD;
	wTensaoMaximaAN_W1: WORD;
	wTensaoMaximaAN_W0: WORD;
	wTensaoMaximaBN_W1: WORD;
	wTensaoMaximaBN_W0: WORD;
	wTensaoMaximaCN_W1: WORD;
	wTensaoMaximaCN_W0: WORD;
	wTensaoMaximaAvgN_W1: WORD;
	wTensaoMaximaAvgN_W0: WORD;
	wPotenciaAtivaTotalMaxima_W1: WORD;
	wPotenciaAtivaTotalMaxima_W0: WORD;
	EnergiaAtivaAcumulada: ConverLintReal;
	EnergiaReativaAcumulada: ConverLintReal;
	EnergiaAparenteAcumulada: ConverLintReal;
END_VAR

(*fCorrenteFaseA:=Valor_Float(wCorrenteFaseA_W0, wCorrenteFaseA_W1);
fCorrenteFaseB:=Valor_Float(wCorrenteFaseB_W0, wCorrenteFaseB_W1);
fCorrenteFaseC:=Valor_Float(wCorrenteFaseC_W0, wCorrenteFaseC_W1);
fCorrenteNeutro:=Valor_Float(wCorrenteNeutro_W0, wCorrenteNeutro_W1);
fCorrenteG:=Valor_Float(wCorrenteG_W0, wCorrenteG_W1);
fCorrenteAvg:=Valor_Float(wCorrenteAvg_W0, wCorrenteAvg_W1);

fTensaoAB:=Valor_Float(WTensaoAB_W0, WTensaoAB_W1);
fTensaoBC:=Valor_Float(wTensaoBC_W0, wTensaoBC_W1);
fTensaoCA:=Valor_Float(wTensaoCA_W0, wTensaoCA_W1);
fTensaoAvgLL:=Valor_Float(wTensaoAvgL_W0, wTensaoAvgL_W1);
fTensaoAN:=Valor_Float(wTensaoAN_W0, wTensaoAN_W1);
fTensaoBN:=Valor_Float(wTensaoBN_W0, wTensaoBN_W1);
fTensaoCN:=Valor_Float(wTensaoCN_W0, wTensaoCN_W1);
fTensaoAvgLN:=Valor_Float(wTensaoAvgN_W0, wTensaoAvgN_W1);

fPotenciaAtivaTotal:=Valor_Float(wPotenciaAtivaTotal_W0, wPotenciaAtivaTotal_W1);

fFatorPotenciaTotal:=Valor_Float(wFatorPotenciaTotal_W0, wFatorPotenciaTotal_W1);

fFrequencia:=Valor_Float(wFrequencia_W0, wFrequencia_W1);

fUltimaDemanda:=Valor_Float(wUltimaDemanda_W0, wUltimaDemanda_W1);
fAtualDemanda:=Valor_Float(wAtualDemanda_W0, wAtualDemanda_W1);
fPrevisaoDemanda:=Valor_Float(wPrevisaoDemanda_W0, wPrevisaoDemanda_W1);
fPicoDemanda:=Valor_Float(wPicoDemanda_W0, wPicoDemanda_W1);
*)

wCorrenteFaseA_MW0 := MOVE(wCorrenteFaseA_W0);
wCorrenteFaseA_MW1 := MOVE(wCorrenteFaseA_W1);
wCorrenteFaseB_MW0 := MOVE(wCorrenteFaseB_W0);
wCorrenteFaseB_MW1 := MOVE(wCorrenteFaseB_W1);
wCorrenteFaseC_MW0 := MOVE(wCorrenteFaseC_W0);
wCorrenteFaseC_MW1 := MOVE(wCorrenteFaseC_W1);
wCorrenteNeutro_MW0	:= MOVE(wCorrenteNeutro_W0);
wCorrenteNeutro_MW1	:= MOVE(wCorrenteNeutro_W1);
wCorrenteG_MW0	:= MOVE(wCorrenteG_W0);
wCorrenteG_MW1	:= MOVE(wCorrenteG_W1);
wCorrenteAvg_MW0	:= MOVE(wCorrenteAvg_W0);
wCorrenteAvg_MW1	:= MOVE(wCorrenteAvg_W1);

wTensaoAB_MW0	:= MOVE(wTensaoAB_W0);
wTensaoAB_MW1	:= MOVE(wTensaoAB_W1);
wTensaoBC_MW0	:= MOVE(wTensaoBC_W0);
wTensaoBC_MW1	:= MOVE(wTensaoBC_W1);
wTensaoCA_MW0	:= MOVE(wTensaoCA_W0);
wTensaoCA_MW1	:= MOVE(wTensaoCA_W1);
wTensaoAvgL_MW0	:= MOVE(wTensaoAvgL_W0);
wTensaoAvgL_MW1	:= MOVE(wTensaoAvgL_W1);
wTensaoAN_MW0	:= MOVE(wTensaoAN_W0);
wTensaoAN_MW1	:= MOVE(wTensaoAN_W1);
wTensaoBN_MW0	:= MOVE(wTensaoBN_W0);
wTensaoBN_MW1	:= MOVE(wTensaoBN_W1);
wTensaoCN_MW0	:= MOVE(wTensaoCN_W0);
wTensaoCN_MW1	:= MOVE(wTensaoCN_W1);
wTensaoAvgN_MW0	:= MOVE(wTensaoAvgN_W0);
wTensaoAvgN_MW1	:= MOVE(wTensaoAvgN_W1);

wPotenciaAtivaTotal_MW0	:= MOVE(wPotenciaAtivaTotal_W0);
wPotenciaAtivaTotal_MW1	:= MOVE(wPotenciaAtivaTotal_W1);

wFatorPotenciaTotal_MW0	:= MOVE(wFatorPotenciaTotal_W0);
wFatorPotenciaTotal_MW1	:= MOVE(wFatorPotenciaTotal_W1);

wFrequencia_MW0	:= MOVE(wFrequencia_W0);
wFrequencia_MW1	:= MOVE(wFrequencia_W1);

wUltimaDemanda_MW0 := MOVE(wUltimaDemanda_W0);
wUltimaDemanda_MW1 := MOVE(wUltimaDemanda_W1);
wAtualDemanda_MW0 := MOVE(wAtualDemanda_W0);
wAtualDemanda_MW1 := MOVE(wAtualDemanda_W1);
wPrevisaoDemanda_MW0 := MOVE(wPrevisaoDemanda_W0);
wPrevisaoDemanda_MW1 := MOVE(wPrevisaoDemanda_W1);
wPicoDemanda_MW0 := MOVE(wPicoDemanda_W0);
wPicoDemanda_MW1 := MOVE(wPicoDemanda_W1);

// Valores INT64
//Consumo Energia Ativa
wEnergiaAtivaAcumulada_MW0_High:= MOVE(wEnergiaAtivaAcumulada_W0_High);
wEnergiaAtivaAcumulada_MW1_High:= MOVE(wEnergiaAtivaAcumulada_W1_High);
wEnergiaAtivaAcumulada_MW0_Low:= MOVE(wEnergiaAtivaAcumulada_W0_Low);
wEnergiaAtivaAcumulada_MW1_Low:= MOVE(wEnergiaAtivaAcumulada_W1_Low);

EnergiaAtivaAcumulada(dValorLow:= dEnergiaAtivaAcumulada_D_Low, dValorHigh:= dEnergiaAtivaAcumulada_D_High, lValorOut=> lEnergiaAtivaAcumulada, rValorOut=>fEnergiaAtivaAcumulada );

//Consumo Energia Reativa
wEnergiaReativaAcumulada_MW0_High:= MOVE(wEnergiaReativaAcumulada_W0_High);
wEnergiaReativaAcumulada_MW1_High:= MOVE(wEnergiaReativaAcumulada_W1_High);
wEnergiaReativaAcumulada_MW0_Low:= MOVE(wEnergiaReativaAcumulada_W0_Low);
wEnergiaReativaAcumulada_MW1_Low:= MOVE(wEnergiaReativaAcumulada_W1_Low);

EnergiaReativaAcumulada(dValorLow:= dEnergiaReativaAcumulada_D_Low, dValorHigh:= dEnergiaReativaAcumulada_D_High, lValorOut=> lEnergiaReativaAcumulada, rValorOut=>fEnergiaReativaAcumulada );

//Consumo Energia Aparente
wEnergiaAparenteAcumulada_MW0_High:= MOVE(wEnergiaAparenteAcumulada_W0_High);
wEnergiaAparenteAcumulada_MW1_High:= MOVE(wEnergiaAparenteAcumulada_W1_High);
wEnergiaAparenteAcumulada_MW0_Low:= MOVE(wEnergiaAparenteAcumulada_W0_Low);
wEnergiaAparenteAcumulada_MW1_Low:= MOVE(wEnergiaAparenteAcumulada_W1_Low);

EnergiaAparenteAcumulada(dValorLow:= dEnergiaAparenteAcumulada_D_Low, dValorHigh:= dEnergiaAparenteAcumulada_D_High, lValorOut=> lEnergiaAparenteAcumulada, rValorOut=>fEnergiaAparenteAcumulada );

// MÁXIMOS
fCorrenteMaximaFaseA:=Valor_Float(wCorrenteMaximaFaseA_W0, wCorrenteMaximaFaseA_W1);
fCorrenteMaximaFaseB:=Valor_Float(wCorrenteMaximaFaseB_W0, wCorrenteMaximaFaseB_W1);
fCorrenteMaximaFaseC:=Valor_Float(wCorrenteMaximaFaseC_W0, wCorrenteMaximaFaseC_W1);
fCorrenteMaximaNeutro:=Valor_Float(wCorrenteMaximaNeutro_W0, wCorrenteMaximaNeutro_W1);
fCorrenteMaximaG:=Valor_Float(wCorrenteMaximaG_W0, wCorrenteMaximaG_W1);
fCorrenteMaximaAvg:=Valor_Float(wCorrenteMaximaAvg_W0, wCorrenteMaximaAvg_W1);

fTensaoMaximaAB:=Valor_Float(wTensaoMaximaAB_W0,wTensaoMaximaAB_W1);
fTensaoMaximaBC:=Valor_Float(wTensaoMaximaBC_W0,wTensaoMaximaBC_W1);
fTensaoMaximaCA:=Valor_Float(wTensaoMaximaCA_W0,wTensaoMaximaCA_W1);
fTensaoMaximaAvgL:=Valor_Float(wTensaoMaximaAvgL_W0,wTensaoMaximaAvgL_W1);
fTensaoMaximaAN:=Valor_Float(wTensaoMaximaAN_W0,wTensaoMaximaAN_W1);
fTensaoMaximaBN:=Valor_Float(wTensaoMaximaBN_W0,wTensaoMaximaBN_W1);
fTensaoMaximaCN:=Valor_Float(wTensaoMaximaCN_W0,wTensaoMaximaCN_W1);
fTensaoMaximaAvgN:=Valor_Float(wTensaoMaximaAvgN_W0,wTensaoMaximaAvgL_W1);

fPotenciaAtivaTotalMaxima:=Valor_Float(wPotenciaAtivaTotalMaxima_W0,wPotenciaAtivaTotalMaxima_W1);

(*------------------------------------------------------------------------
fFatorPotenciaTotal:= WORD_AS_REAL (wFatorPotenciaTotal_W1,wFatorPotenciaTotal_W0);

fUltimaDemanda:=WORD_AS_REAL(wUltimaDemanda_W1, wUltimaDemanda_W0);
fAtualDemanda:=WORD_AS_REAL(wAtualDemanda_W1, wAtualDemanda_W0);
fPrevisaoDemanda:=WORD_AS_REAL(wPrevisaoDemanda_W1, wPrevisaoDemanda_W0);
fPicoDemanda:=WORD_AS_REAL(wPicoDemanda_W1, wPicoDemanda_W0);
*)

(* ---- TesteEnergia.prg.st ---- *)
PROGRAM TesteEnergia
VAR
	///Consumo Ativo
	ContadorConsumo: CTU;
	xContadorCu: BOOL;
	xContadorRst: BOOL;
	///wContadorCv				: WORD;
	ClockConsumo: BLINK;
	xClockConsumoIn: BOOL;
	BloqContador: BOOL;
	rConsumoEnergiaReal: REAL;
	///Consumo Reativo
	ContadorConsumoVa: CTU;
	xContadorVaCu: BOOL;
	xContadorVaRst: BOOL;
	///wContadorCv				: WORD;
	ClockConsumoVa: BLINK;
	xClockConsumoVaIn: BOOL;
	BloqContadorVa: BOOL;
	rConsumoEnergiaReativaReal: REAL;
	TonHabilit: TON;
	xTonHabilitIn: BOOL;
	xTonHabilitQ: BOOL;
	xIntervaloFPont: BOOL;
	xIntervaloPont: BOOL;
	LeituraDemand: REAL;
	///xFimMes: BOOL;
	///
	///
	///	rMesFatura: INT;
	///	rAnoFatura: INT;
	///parametros permanentes
	PassoInterval: INT;
	xSelecaoIntervalo: BOOL;
	wContadorCv: WORD;
	wContadorVaCv: WORD;
	///Energia Ativa
	rConsumoInicialFPont: REAL;
	rConsumoInstantaneoFPont: REAL;
	rConsumoAcumuladoFPont: REAL;
	rConsumoInstantAcumFPont: REAL;
	rConsumoFPont: REAL;
	rConsumoInicialPont: REAL;
	rConsumoInstantaneoPont: REAL;
	rConsumoAcumuladoPont: REAL;
	rConsumoInstantAcumPont: REAL;
	rConsumoPont: REAL;
	///Energia Reativa
	rConsumoInicialFPontVa: REAL;
	rConsumoInstantaneoFPontVa: REAL;
	rConsumoAcumuladoFPontVa: REAL;
	rConsumoInstantAcumFPontVa: REAL;
	rConsumoFPontVa: REAL;
	rConsumoInicialPontVa: REAL;
	rConsumoInstantaneoPontVa: REAL;
	rConsumoAcumuladoPontVa: REAL;
	rConsumoInstantAcumPontVa: REAL;
	rConsumoPontVa: REAL;
	///Demanda
	rDemandMaxima: REAL;
	rDemandInstantanea: REAL;
	xHabilitaPm: BOOL;
END_VAR

rDemandInstantanea:=LeituraDemand;
IF rDemandInstantanea>rDemandMaxima AND NOT xHabilitaPm THEN
	rDemandMaxima:=rDemandInstantanea;
END_IF

(*IF xFimMes THEN
	rMesFatura:=rMesFatura;
	rAnoFatura:=rAnoFatura;
	xFechaFatura:=1;
	xFimMes:=FALSE;
	xHabilitaPm:=TRUE;
END_IF

IF xFaturaFechada=1 THEN
	xContadorRst:=TRUE;
END_IF*)

ClockConsumo.ENABLE:= NOT xHabilitaPm;
ClockConsumoVa.ENABLE:= NOT xHabilitaPm;
//Consumo Ativo

ClockConsumo(ENABLE:= , TIMELOW:=T#1S , TIMEHIGH:=T#1S , OUT=> xContadorCu);

IF xContadorCu AND NOT BloqContador THEN
	wContadorCv:=wContadorCv+1;
	BloqContador:=TRUE;
END_IF

IF NOT xContadorCu  THEN
	BloqContador:=FALSE;
END_IF

rConsumoEnergiaReal:= WORD_TO_REAL ((wContadorCv))/10;

//Consumo Reativo
ClockConsumoVa(ENABLE:= , TIMELOW:=T#3S , TIMEHIGH:=T#3S , OUT=> xContadorVaCu);

IF xContadorVaCu AND NOT BloqContadorVa THEN
	wContadorVaCv:=wContadorVaCv+1;
	BloqContadorVa:=TRUE;
END_IF

IF NOT xContadorVaCu  THEN
	BloqContadorVa:=FALSE;
END_IF

rConsumoEnergiaReativaReal:= WORD_TO_REAL ((wContadorVaCv))/10;

/////////////////////////////////////////////////////////////

IF xSelecaoIntervalo THEN
	xIntervaloPont:=TRUE;
	xIntervaloFPont:=FALSE;
ELSE
	xIntervaloFPont:=TRUE;
	xIntervaloPont:=FALSE;
END_IF

xTonHabilitIn:=TRUE;
TonHabilit(IN:=xTonHabilitIn , PT:=T#300MS , Q=> xTonHabilitQ, ET=> );

CASE PassoInterval OF

		0: 	IF xIntervaloFPont AND xTonHabilitQ THEN
				PassoInterval:=5;
			END_IF
			IF xIntervaloPont AND xTonHabilitQ THEN
				PassoInterval:=50;
			END_IF

		5:	rConsumoInicialFPont:=rConsumoEnergiaReal;(*Ativa*)
			rConsumoInicialFPontVa:=rConsumoEnergiaReativaReal;(*Reativa*)
			PassoInterval:=10;

		10:	rConsumoInstantaneoFPont:=rConsumoEnergiaReal-rConsumoInicialFPont;(*Ativa*)
			rConsumoInstantAcumFPont:=rConsumoAcumuladoFPont+rConsumoInstantaneoFPont;(*Ativa*)
			rConsumoInstantaneoFPontVa:=rConsumoEnergiaReativaReal-rConsumoInicialFPontVa;(*Reativa*)
			rConsumoInstantAcumFPontVa:=rConsumoAcumuladoFPontVa+rConsumoInstantaneoFPontVa;(*Reativa*)
			IF (NOT xIntervaloFPont OR (xFechaFatura=1)) AND xTonHabilitQ THEN
				PassoInterval:=15;
			END_IF

		15:	rConsumoFPont:=rConsumoInstantaneoFPont;(*Ativo*)
			rConsumoAcumuladoFPont:=rConsumoInstantAcumFPont;(*Ativo*)
			rConsumoFPontVa:=rConsumoInstantaneoFPontVa;(*Reativo*)
			rConsumoAcumuladoFPontVa:=rConsumoInstantAcumFPontVa;(*Reativo*)
			PassoInterval:=20;

		20:	rConsumoInstantaneoFPont:=0;(*Ativo*)
			rConsumoInstantaneoFPontVa:=0;(*Reativo*)
			PassoInterval:=0;

		50:	rConsumoInicialPont:=rConsumoEnergiaReal;(*Ativo*)
			rConsumoInicialPontVa:=rConsumoEnergiaReativaReal;(*Reativo*)
			PassoInterval:=55;

		55:	rConsumoInstantaneoPont:=rConsumoEnergiaReal-rConsumoInicialPont;(*Ativo*)
			rConsumoInstantAcumPont:=rConsumoAcumuladoPont+rConsumoInstantaneoPont;(*Ativo*)
			rConsumoInstantaneoPontVa:=rConsumoEnergiaReativaReal-rConsumoInicialPontVa;(*Reativo*)
			rConsumoInstantAcumPontVa:=rConsumoAcumuladoPontVa+rConsumoInstantaneoPontVa;(*Reativo*)
			IF (NOT xIntervaloPont OR (xFechaFatura=1))AND xTonHabilitQ THEN
				PassoInterval:=60;
			END_IF

		60:	rConsumoPont:=rConsumoInstantaneoPont;(*Ativo*)
			rConsumoAcumuladoPont:=rConsumoInstantAcumPont;(*Ativo*)
			rConsumoPontVa:=rConsumoInstantaneoPontVa;(*Reativo*)
			rConsumoAcumuladoPontVa:=rConsumoInstantAcumPontVa;(*Reativo*)
			PassoInterval:=65;

		65:	rConsumoInstantaneoPont:=0;(*Ativo*)
			rConsumoInstantaneoPont:=0;(*Reativo*)
			PassoInterval:=0;
END_CASE

IF xContadorRst THEN
	rConsumoInicialFPont	:=0 ;
	rConsumoInstantaneoFPont:=0 ;
	rConsumoAcumuladoFPont	:=0 ;
	rConsumoInstantAcumFPont:=0 ;
	rConsumoFPont			:=0 ;

	rConsumoInicialPont		:=0 ;
	rConsumoInstantaneoPont	:=0 ;
	rConsumoAcumuladoPont	:=0 ;
	rConsumoInstantAcumPont	:=0 ;
	rConsumoPont			:=0 ;
	wContadorCv				:=0 ;
	xContadorRst			:=0 ;

	rConsumoInicialFPontVa	:=0 ;
	rConsumoInstantaneoFPontVa:=0 ;
	rConsumoAcumuladoFPontVa	:=0 ;
	rConsumoInstantAcumFPontVa:=0 ;
	rConsumoFPontVa			:=0 ;

	rConsumoInicialPontVa		:=0 ;
	rConsumoInstantaneoPontVa	:=0 ;
	rConsumoAcumuladoPontVa	:=0 ;
	rConsumoInstantAcumPontVa	:=0 ;
	rConsumoPontVa			:=0 ;
	wContadorVaCv				:=0 ;
	xContadorVaRst			:=0 ;

	rDemandMaxima				:=0;
	rDemandInstantanea			:=0;
	xHabilitaPm					:=FALSE;
	//xFaturaFechada				:=0;
	xContadorRst				:=FALSE;
END_IF
